FUNCTION F_IsBusy : BOOL;
VAR_INPUT
	Feedback : I_CommandFeedback;
END_VAR

IF Feedback <> 0 AND_THEN Feedback.Busy THEN
	F_IsBusy := TRUE;
END_IF

END_FUNCTION

(* stored: Version 1.1.0.1, ProductVersion 3.1.4024.12
   POU F_IsBusy: Id {3ff8e7bf-f005-02d8-3c7f-1cbbbdf0aa53}, SpecialFunc None *)
